FUNCTION_BLOCK Five_State_Actuator_CAT (* Composite Function Block Type *)
  (* Standard: 61499-2 *)
  (* Version 0.0, 10/7/2025, Schneider Electric, template *)
  PACKAGE Main;
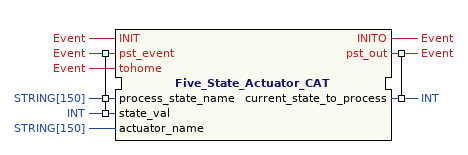
  EVENT_INPUT
    INIT; (* Initialization Request *)
    pst_event WITH process_state_name, state_val; (* Normal Execution Request *)
    tohome;
  END_EVENT
  EVENT_OUTPUT
    INITO; (* Initialization Confirm *)
    pst_out WITH current_state_to_process; (* Execution Confirmation *)
  END_EVENT
  VAR_INPUT
    process_state_name : STRING[150];
    state_val : INT;
    actuator_name : STRING[150];
  END_VAR
  VAR_OUTPUT
    current_state_to_process : INT; (* Output event qualifier *)
  END_VAR
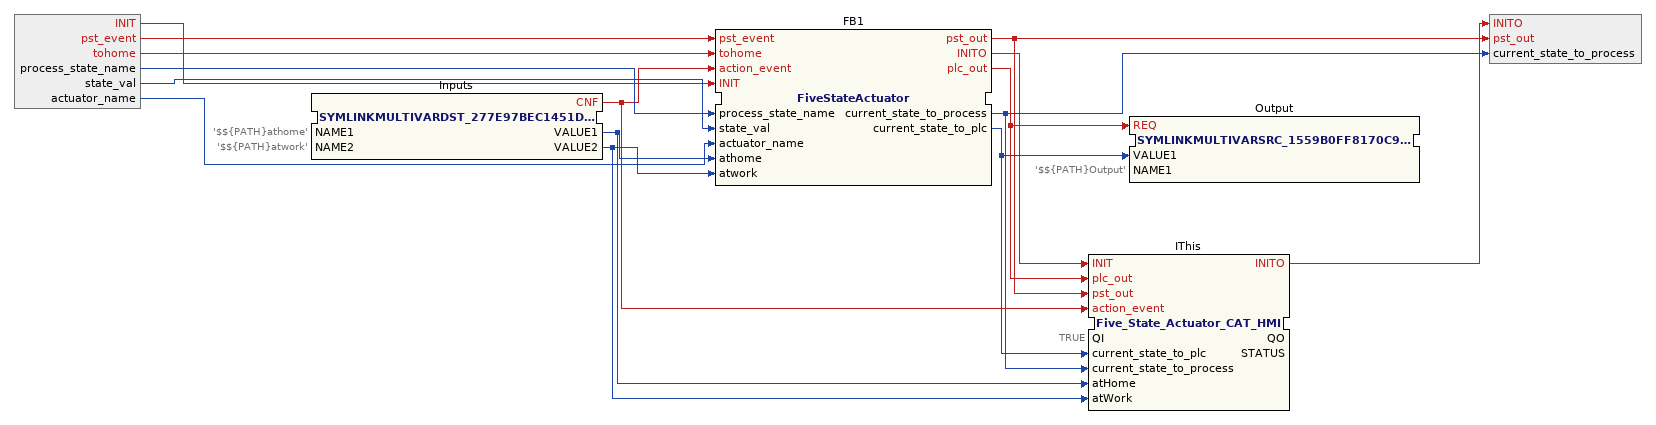
  FBS
    FB1 : FiveStateActuator;
    IThis : Five_State_Actuator_CAT_HMI(QI := TRUE);
    Inputs : SYMLINKMULTIVARDST_277E97BEC1451D2C(NAME1 := '$${PATH}athome', NAME2 := '$${PATH}atwork'); {SET_ATTRIBUTE(Configuration.GenericFBType.InterfaceParams, Runtime.System#I:=2;VALUE${I$}:BOOL,BOOL)}
    Output : SYMLINKMULTIVARSRC_1559B0FF8170C9BA0(NAME1 := '$${PATH}Output'); {SET_ATTRIBUTE(Configuration.GenericFBType.InterfaceParams, Runtime.System#I:=1;VALUE${I$}:BOOL)}
  END_FBS
  EVENT_CONNECTIONS
    pst_event TO FB1.pst_event;
    tohome TO FB1.tohome;
    FB1.pst_out TO pst_out;
    Inputs.CNF TO FB1.action_event;
    INIT TO FB1.INIT;
    FB1.INITO TO IThis.INIT;
    FB1.plc_out TO IThis.plc_out;
    FB1.pst_out TO IThis.pst_out;
    Inputs.CNF TO IThis.action_event;
    IThis.INITO TO INITO;
    FB1.plc_out TO Output.REQ;
  END_CONNECTIONS
  DATA_CONNECTIONS
    process_state_name TO FB1.process_state_name;
    state_val TO FB1.state_val;
    actuator_name TO FB1.actuator_name;
    FB1.current_state_to_process TO current_state_to_process;
    Inputs.VALUE1 TO FB1.athome;
    Inputs.VALUE2 TO FB1.atwork;
    FB1.current_state_to_plc TO IThis.current_state_to_plc;
    FB1.current_state_to_process TO IThis.current_state_to_process;
    Inputs.VALUE1 TO IThis.atHome;
    Inputs.VALUE2 TO IThis.atWork;
    FB1.current_state_to_plc TO Output.VALUE1;
  END_CONNECTIONS
END_FUNCTION_BLOCK
